// TIA Portal V20 export
DATA_BLOCK "SomeInstance"   // DB4
// stored: InstanceOfName SomeFB, InstanceOfType FB
"SomeFB"
   // VAR
   //    Flag : Bool;
   // END_VAR
BEGIN
END_DATA_BLOCK
